// Mitsubishi GX Works2 project: 실린더 제어하기 엑셀 데이터로 저장2-1 0923   PLC: Q03UDV

PROGRAM MAIN
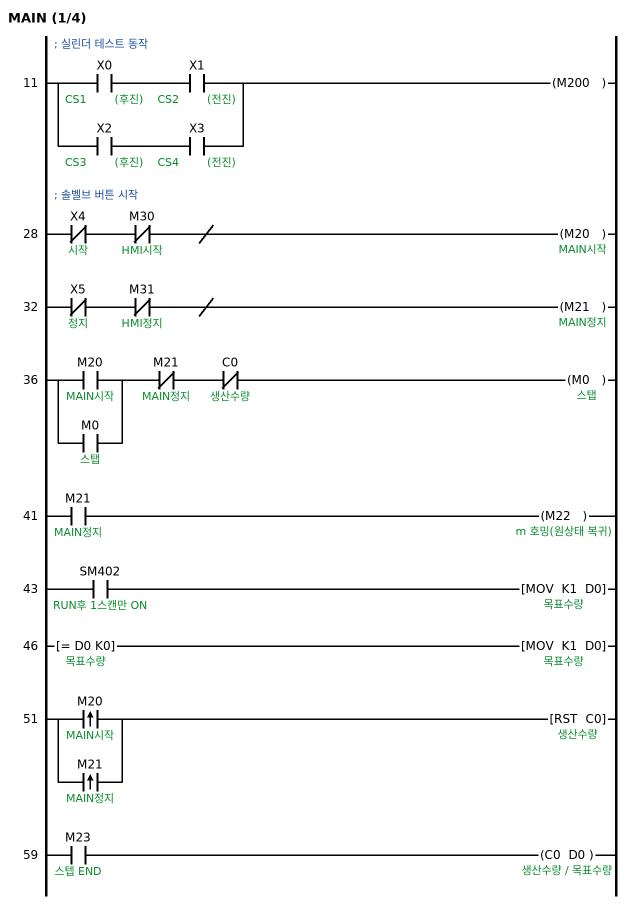
; 실린더 테스트 동작
11    LD      X0  ; CS1        (후진)
      AND     X1  ; CS2        (전진)
      LD      X2  ; CS3        (후진)
      AND     X3  ; CS4        (전진)
      ORB
      OUT     M200
; 솔벨브 버튼 시작
28    LDI     X4  ; 시작
      ANI     M30  ; HMI시작
      INV
      OUT     M20  ; MAIN시작
32    LDI     X5  ; 정지
      ANI     M31  ; HMI정지
      INV
      OUT     M21  ; MAIN정지
36    LD      M20  ; MAIN시작
      OR      M0  ; 스탭
      ANI     M21  ; MAIN정지
      ANI     C0  ; 생산수량
      OUT     M0  ; 스탭
41    LD      M21  ; MAIN정지
      OUT     M22  ; m 호밍(원상태 복귀)
43    LD      SM402  ; RUN후 1스캔만 ON
      MOV     K1 D0  ; 목표수량
46    LD=     D0 K0  ; 목표수량
      MOV     K1 D0
51    LDP     M20  ; MAIN시작
      ORP     M21  ; MAIN정지
      RST     C0  ; 생산수량
59    LD      M23  ; 스텝 END
      OUT     C0 D0  ; 생산수량 / 목표수량
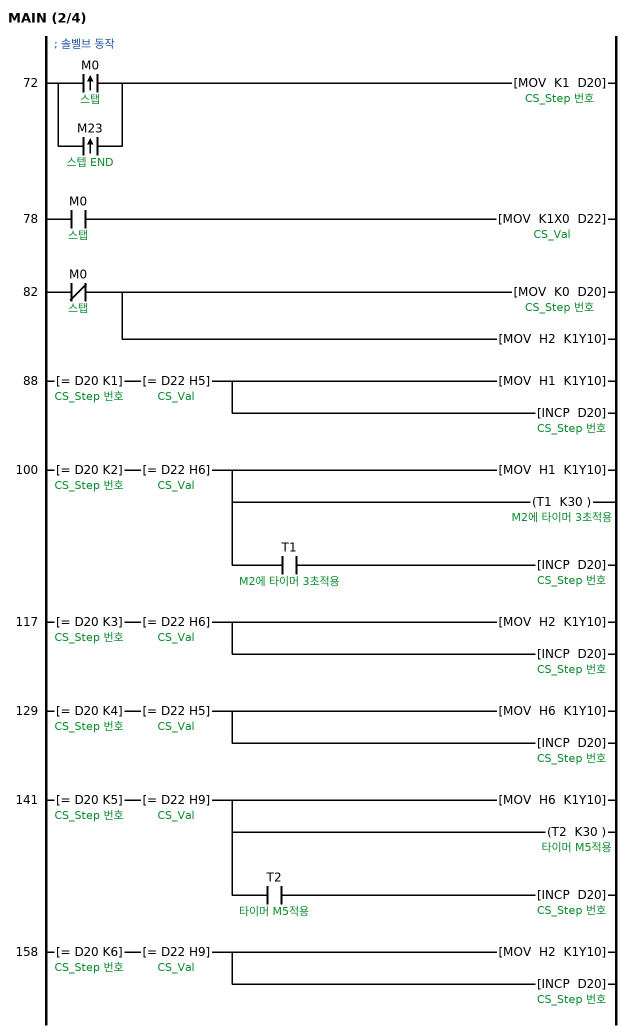
; 솔벨브 동작
72    LDP     M0  ; 스탭
      ORP     M23  ; 스텝 END
      MOV     K1 D20  ; CS_Step 번호
78    LD      M0  ; 스탭
      MOV     K1X0 D22  ; CS_Val
82    LDI     M0  ; 스탭
      MOV     K0 D20
      MOV     H2 K1Y10  ; 양솔전진
88    LD=     D20 K1  ; CS_Step 번호
      AND=    D22 H5  ; CS_Val
      MOV     H1 K1Y10
      INCP    D20
100   LD=     D20 K2  ; CS_Step 번호
      AND=    D22 H6  ; CS_Val
      MOV     H1 K1Y10
      OUT     T1 K30  ; M2에 타이머 3초적용
      AND     T1  ; M2에 타이머 3초적용
      INCP    D20
117   LD=     D20 K3  ; CS_Step 번호
      AND=    D22 H6  ; CS_Val
      MOV     H2 K1Y10
      INCP    D20
129   LD=     D20 K4  ; CS_Step 번호
      AND=    D22 H5  ; CS_Val
      MOV     H6 K1Y10
      INCP    D20
141   LD=     D20 K5  ; CS_Step 번호
      AND=    D22 H9  ; CS_Val
      MOV     H6 K1Y10
      OUT     T2 K30  ; 타이머 M5적용
      AND     T2  ; 타이머 M5적용
      INCP    D20
158   LD=     D20 K6  ; CS_Step 번호
      AND=    D22 H9  ; CS_Val
      MOV     H2 K1Y10
      INCP    D20
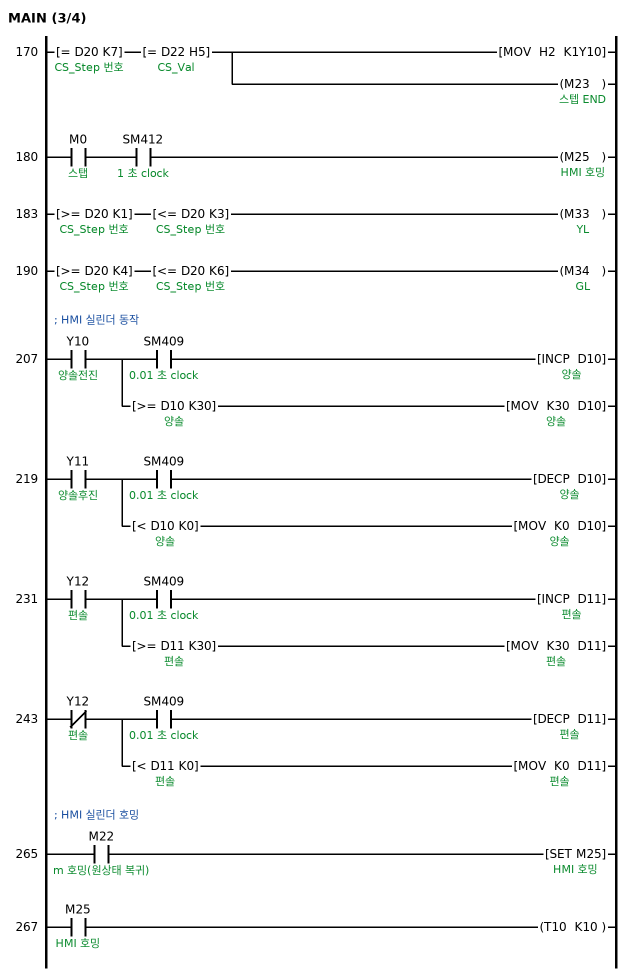
170   LD=     D20 K7  ; CS_Step 번호
      AND=    D22 H5  ; CS_Val
      MOV     H2 K1Y10
      OUT     M23  ; 스텝 END
180   LD      M0  ; 스탭
      AND     SM412  ; 1 초 clock
      OUT     M25  ; HMI 호밍
183   LD>=    D20 K1  ; CS_Step 번호
      AND<=   D20 K3  ; CS_Step 번호
      OUT     M33  ; YL
190   LD>=    D20 K4  ; CS_Step 번호
      AND<=   D20 K6  ; CS_Step 번호
      OUT     M34  ; GL
; HMI 실린더 동작
207   LD      Y10  ; 양솔전진
      MPS
      AND     SM409  ; 0.01 초 clock
      INCP    D10  ; 양솔
      MPP
      AND>=   D10 K30  ; 양솔
      MOV     K30 D10
219   LD      Y11  ; 양솔후진
      MPS
      AND     SM409  ; 0.01 초 clock
      DECP    D10
      MPP
      AND<    D10 K0  ; 양솔
      MOV     K0 D10
231   LD      Y12  ; 편솔
      MPS
      AND     SM409  ; 0.01 초 clock
      INCP    D11  ; 편솔
      MPP
      AND>=   D11 K30  ; 편솔
      MOV     K30 D11
243   LDI     Y12  ; 편솔
      MPS
      AND     SM409  ; 0.01 초 clock
      DECP    D11
      MPP
      AND<    D11 K0  ; 편솔
      MOV     K0 D11
; HMI 실린더 호밍
265   LD      M22  ; m 호밍(원상태 복귀)
      SET     M25  ; HMI 호밍
267   LD      M25  ; HMI 호밍
      OUT     T10 K10
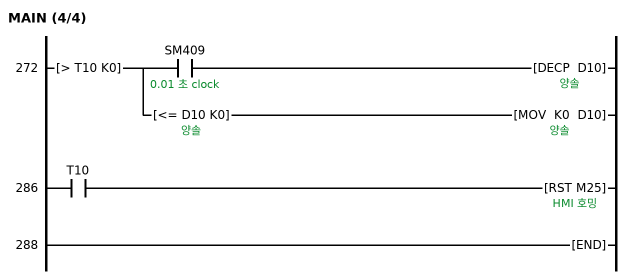
272   LD>     T10 K0
      MPS
      AND     SM409  ; 0.01 초 clock
      DECP    D10
      MPP
      AND<=   D10 K0  ; 양솔
      MOV     K0 D10
286   LD      T10
      RST     M25  ; HMI 호밍
288   END
END_PROGRAM

// device comments not shown above
Y13  ; 부저
M1  ; 스탭 1
M2  ; 스탭 2
M3  ; 스탭 3
M4  ; 스텝 4
M5  ; 스텝5
M6  ; 스텝6
M7  ; 스텝7
M24  ; M_부저
M32  ; RL
D24  ; Sol_Val
T0  ; 타이머
